Fanuc KAREL source: kb00109.KL

-- PROVISIONAL review KL for V1013-1; original PC SHA256 283cd0d265cfb2b8fb3297284772079f744611806a3254aa6d624f589d8495df
-- Incomplete behavior may be omitted. Consult companion uncertainty JSON. Do not deploy.
PROGRAM KB00109
%NOLOCKGROUP
-- UNRESOLVED_DECL P1 type=000101
-- UNRESOLVED_DECL RESULT type=000101
BEGIN
  -- UNRESOLVED_PC offsets 5-32; opcodes 27,22,1C,76,7E,4A
  -- UNRESOLVED_PC offsets 37-41; opcodes 7F
END KB00109
